# EPICS substitutions: ek9000App/Db/EL2798.substitutions
file EL2798.template
{       pattern
        {
                TERMINAL,

        }
        {
        }
}
